FUNCTION_BLOCK Fan
VAR_INPUT
END_VAR
VAR_OUTPUT
END_VAR
VAR
	xOutputAddress AT %I* : BIT;
	bPowerStatus : BOOL;
END_VAR

METHOD FB_init : BOOL
VAR_INPUT
	bInitRetains : BOOL; // if TRUE, the retain variables are initialized (warm start / cold start)
	bInCopyCode : BOOL;  // if TRUE, the instance afterwards gets moved into the copy code (online change)
END_VAR
END_METHOD

METHOD powerOff : BOOL
VAR_INPUT
END_VAR
END_METHOD

METHOD powerOn : BOOL
VAR_INPUT
END_VAR
END_METHOD

PROPERTY PUBLIC powerStatus : BOOL
GET
powerStatus := bPowerStatus;
END_GET
END_PROPERTY

END_FUNCTION_BLOCK

(* stored: Version 1.1.0.1, ProductVersion 3.1.4024.12
   POU Fan: Id {95480810-6c45-406d-a0b3-81d20a535b10}, SpecialFunc None
   Method FB_init: Id {4833a7f0-075c-4b92-aeed-a732432b88a7}
   Method powerOff: Id {a3845553-ff17-4947-b43e-e8b2f09ad26f}
   Method powerOn: Id {28b2fa98-3340-4b57-8e91-5ef09854043c}
   Property powerStatus: Id {e4b16a19-1d7c-4798-ba7c-cc208ec70e8d}
   Get Get: Id {bf8b66fa-7660-4047-a96f-836253c43622} *)
